{attribute 'linkalways'} 
{attribute 'no_explicit_call' := 'This FB is a CLASS and must be accessed using methods or properties'}
{attribute 'enable_dynamic_creation'}
FUNCTION_BLOCK FINAL MOD_WORD EXTENDS Node
VAR
	in1 : _WORD(0);
	in2 : _WORD(0);
	out : _WORD(0);
END_VAR

METHOD PUBLIC Clone : I_Node
VAR
	pNode : POINTER TO MOD_WORD;
END_VAR
pNode := __NEW(MOD_WORD);
Clone := pNode^;
END_METHOD

METHOD FB_init : BOOL
VAR_INPUT
	bInitRetains : BOOL; // if TRUE, the retain variables are initialized (warm start / cold start)
	bInCopyCode : BOOL;  // if TRUE, the instance afterwards gets moved into the copy code (online change)
END_VAR
AddInput('in1',THIS^.in1);
AddInput('in2',THIS^.in2);
AddOutput('out', THIS^.out);
END_METHOD

METHOD PROTECTED OnExecute
VAR
END_VAR
out.Value := in1.Value MOD in2.Value;
END_METHOD

END_FUNCTION_BLOCK

(* stored: Version 1.1.0.1, ProductVersion 3.1.4024.15
   POU MOD_WORD: Id {7a8fec7c-6ef6-4825-bc8a-33baa45e2380}, SpecialFunc None
   Folder Constructor: Id {ce405ec7-4fd4-4b55-a00a-3bbaf6964904}
   Method Clone: Id {93bc1586-d3b8-4d24-9ccd-2cea9bfec236}
   Method FB_init: Id {ea3a5b42-1456-402c-ad02-7d69991acbd7}
   Method OnExecute: Id {067d4d8e-4a37-4ce3-94a1-b2f5529a1182} *)
